FUNCTION_BLOCK ExtControlBehaviour IMPLEMENTS I_Cyclic
VAR
	ThisMover : I_XtsMover;
END_VAR

METHOD PUBLIC  Cycle : HRESULT
VAR_INPUT
END_VAR
END_METHOD

METHOD Disable : BOOL
VAR_INPUT
END_VAR
Disable := SUCCEEDED(ThisMover.DisableMover());
END_METHOD

METHOD Enable : BOOL
VAR_INPUT
END_VAR
Enable := SUCCEEDED(ThisMover.EnableMover());
END_METHOD

METHOD Halt : BOOL
VAR_INPUT
END_VAR
Halt := SUCCEEDED(thisMover.HaltAxis());
END_METHOD

METHOD MoveTo : BOOL
VAR_INPUT
	Position : LREAL;
	Velocity : LREAL;
END_VAR
MoveTo := SUCCEEDED(ThisMover.MoveTo(RequiredPosition := Position,
									MoveVelocity := Velocity,
									NonModuloMove := FALSE));
END_METHOD

PROPERTY MyMover : I_XtsMover
GET
MyMover := ThisMover;
END_GET
SET
ThisMover := MyMover;
END_SET
END_PROPERTY

METHOD Reset : BOOL
VAR_INPUT
END_VAR
Reset := SUCCEEDED(ThisMover.Reset());
END_METHOD

END_FUNCTION_BLOCK

(* stored: Version 1.1.0.1
   POU ExtControlBehaviour: Id {d3f2ac87-b8f7-4911-b9c2-b9baff5eb1c4}, SpecialFunc None
   Method Cycle: Id {8888b623-da21-4226-add6-1f1bd1a51781}
   Method Disable: Id {de056d5c-7619-4cd3-985e-6a0d3f8440cf}
   Method Enable: Id {fc9ca77d-9c21-42b3-a164-3c3fa5410e23}
   Method Halt: Id {e8567e91-73af-4e94-abd4-838ab80ff80a}
   Method MoveTo: Id {468f93df-df4c-4d07-b983-c9e7bb93f621}
   Property MyMover: Id {a5c868b0-cac0-4f55-bd66-8ef755b79feb}
   Get Get: Id {587907ca-a173-4213-9ae5-405c4a27d931}
   Set Set: Id {61ecbb90-d62b-4e06-b9a5-e3c58bf4d7f4}
   Method Reset: Id {bd85c3c4-76d3-46ae-9b7a-d256e0218e53} *)
